PROGRAM AP_V2
VAR
	// Bedienparameter
	
	// Prozessparameter
	
	// Skill-Instanziierung
	Skill_R_P2P			:Skill_Position_anfahren;
	Skill_R_Ausrichten	:Skill_Position_anfahren_erweitert;
	Skill_G_P2P			:Skill_Greifer_Pos_Anfahren;
	
	// Sequenz-Instanziierung
	Seq_Get_Teil		:Seq_Teile_Hohlen;
	
	
END_VAR

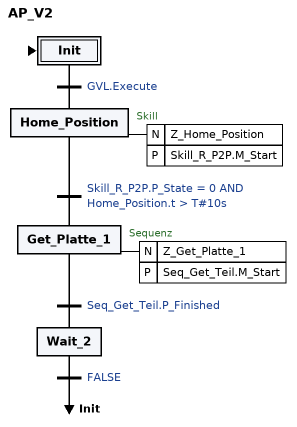
INITIAL_STEP Init:
END_STEP
TRANSITION FROM Init TO Home_Position
    := GVL.Execute;
END_TRANSITION
// Skill
STEP Home_Position:
    Z_Home_Position(N);
    Skill_R_P2P.M_Start(P);
END_STEP
TRANSITION FROM Home_Position TO Get_Platte_1
    := Skill_R_P2P.P_State = 0 AND Home_Position.t > T#10s;
END_TRANSITION
// Sequenz
STEP Get_Platte_1:
    Z_Get_Platte_1(N);
    Seq_Get_Teil.M_Start(P);
END_STEP
TRANSITION FROM Get_Platte_1 TO Wait_2
    := Seq_Get_Teil.P_Finished;
END_TRANSITION
STEP Wait_2:
END_STEP
TRANSITION FROM Wait_2 TO Init
    := FALSE;
END_TRANSITION

ACTION Z_Get_Platte_1:
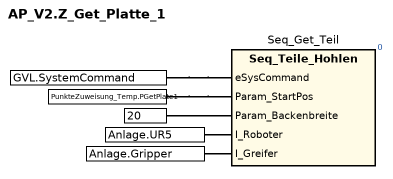
Seq_Get_Teil(
    eSysCommand := GVL.SystemCommand,
    Param_StartPos := PunkteZuweisung_Temp.PGetPlate1,
    Param_Backenbreite := 20,
    I_Roboter := Anlage.UR5,
    I_Greifer := Anlage.Gripper); // Seq_Teile_Hohlen
END_ACTION

ACTION Z_Home_Position:
Skill_R_P2P(eSysCommand := GVL.SystemCommand,
			eSysState := GVL.SystemState,
			Objekt := Anlage.UR5,
			iErrorID => GVL.ErrorID);

Skill_R_P2P.P_RobotParam := PunkteZuweisung_Temp.PHome;
END_ACTION

ACTION Z_Start_Pos:
// Skillaufruf
Skill_R_P2P(eSysCommand := GVL.SystemCommand,
			eSysState := GVL.SystemState,
			Objekt := Anlage.UR5,
			iErrorID => GVL.ErrorID);

		
// Parameterzuweisung	
Skill_R_P2P.P_RobotParam := PunkteZuweisung_Temp.PGetPlate1;
END_ACTION

END_PROGRAM

(* stored: Version 1.1.0.1
   POU AP_V2: Id {ab609da4-227a-4c12-81f2-45f5f4762e7d}, SpecialFunc None
   Folder 01_Zuweisung: Id {bfb8da45-b845-4175-8e26-26b7ccad7777}
   Action Z_Get_Platte_1: Id {bfa14221-1062-449d-b7d4-7340f6f38f81}
   Action Z_Home_Position: Id {49f52d09-a60c-43ff-a568-bdae543b41db}
   Action Z_Start_Pos: Id {7bfdcb5a-449e-4abb-8b01-af39ade7c030} *)
